Universal Robots PolyScope program: square.urp

Program square (installation=default directory=/home/ur/ursim-current/programs createdIn=5.14.0 lastSavedIn=5.14.0 robotSerialNumber=20195299999)
Calibrated DH parameters: a=[0, -0.6127, -0.57155, 0, 0, 0]; d=[0.1807, 0, 0, 0.17415, 0.11985, 0.11655]; alpha=[1.570796, 0, 0, 1.570796, -1.570796, 0]; deltaTheta=[0, 0, 0, 0, 0, 0]
InitVariablesNode
Robot Program (runOnlyOnce=false)
  Script file /home/ur/ursim-current/programs/square.script
    | # UR Square Script
    | 
    | # variables
    | r = 40
    | rep = 2
    | loop = False
    | 
    | # positions (can be defined also as installation variables to keep their last value)
    | global pa = p[0.6, 0, 0.2, 3.14, 0.00, 0.00]
    | global pb = p[0.6, 0.2, 0.2, 3.14, 0.00, 0.00]
    | global pc = p[0.4, 0.2, 0.2, 3.14, 0.00, 0.00]
    | global pd = p[0.4, 0, 0.2, 3.14, 0.00, 0.00]
    | 
    | # functions
    | def move_square():
    |     movel(pa, r=r/1000)
    |     movel(pb, r=r/1000)
    |     movel(pc, r=r/1000)
    |     movel(pd, r=r/1000)
    | end
    | 
    | def square_task():
    |     if loop:
    |         i = 0
    |         while i < rep:
    |             move_square()
    |         end
    |     else:
    |         move_square()
    |    end
    | end
  URCap HMI (Robpod HMI URcap, Robpod Cloud) dataModel(robpod.hmi.selected=/home/ur/ursim-current/programs/square_hmi.hmi, robpod.hmi.stop.main.loop=true)
